// TIA Portal project "Esempio_TCP" (V15.1)

(* hardware
DEVICE "S7-1200 station_2"  S7-1200 Station
   slot 0: "Telaio di montaggio_0"  S7-1200 Rack  Rack  V1.0
   slot 1: "Passivo"  CPU 1214C DC/DC/DC  6ES7 214-1AG40-0XB0  V4.2
DEVICE "S7-1200 station_1"  S7-1200 Station
   slot 0: "Telaio di montaggio_0"  S7-1200 Rack  Rack  V1.0
   slot 1: "Attivo"  CPU 1214C DC/DC/DC  6ES7 214-1AG40-0XB0  V4.2
*)

// ===== PLC "Attivo"  CPU 1214C DC/DC/DC =====

VAR_GLOBAL   // PLC tag table "Tabella delle variabili standard"
   "connetti" AT %I0.0 : Bool;
   "Connesso" AT %M0.0 : Bool;
   "Disconnetti" AT %I0.1 : Bool;
   "invia_dati" AT %I0.2 : Bool;
END_VAR

DATA_BLOCK "Send_block"   // DB4
{ S7_Optimized_Access := 'FALSE' }
VERSION : 0.1
   VAR
      testBool : Bool;
      testInt : Int;
   END_VAR
BEGIN
END_DATA_BLOCK

DATA_BLOCK "Receive_block"   // DB7
{ S7_Optimized_Access := 'FALSE' }
VERSION : 0.1
   VAR
      testBool : Bool;
      testInt : Int;
   END_VAR
BEGIN
END_DATA_BLOCK

// folder: System blocks/Program resources

DATA_BLOCK "Attivo_Connection_DB"   // DB2
{ S7_Optimized_Access := 'TRUE' }
AUTHOR : SIMATIC
FAMILY : MC7Plus
NAME : TC_IP_v4
VERSION : 1.0
// stored: InstanceOfName TCON_IP_v4
"TCON_IP_v4"
BEGIN
   ID := 1;
   InterfaceId := 64;
   RemotePort := 2000;
   ActiveEstablished := true;
   RemoteAddress.ADDR[1] := 192;
   RemoteAddress.ADDR[2] := 168;
   RemoteAddress.ADDR[4] := 2;
END_DATA_BLOCK

// folder: (top level)

ORGANIZATION_BLOCK "Main"   // OB1, LAD, ProgramCycle
TITLE = "Main Program Sweep (Cycle)"
{ S7_Optimized_Access := 'TRUE' }
VERSION : 0.1
   VAR_INPUT
      Initial_Call : Bool;   // Initial call of this OB
      Remanence : Bool;   // =True, if remanent data are available
   END_VAR
   VAR_TEMP
      temp1 : Bool;
      temp2 : Bool;
      temp3 : Bool;
   END_VAR
   VAR_TEMP   // added for the SCL form of the ladder/FBD networks
      _w1 : Bool;
   END_VAR
BEGIN

REGION Network 1
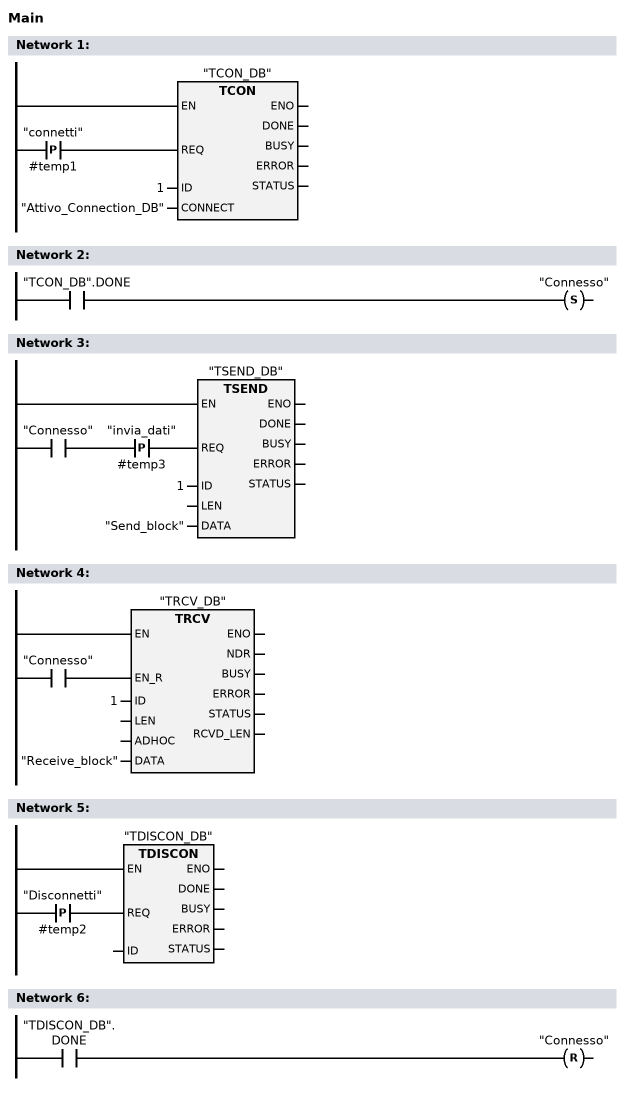
   #_w1 := "connetti" AND NOT #temp1;   // rising edge of "connetti"
   #temp1 := "connetti";
   "TCON_DB"(REQ := #_w1, ID := 1, CONNECT := "Attivo_Connection_DB");   // TCON
END_REGION

REGION Network 2
   RUNG wire#powerrail
      Contact( "TCON_DB".DONE )
      S_Coil( "Connesso" )
   END_RUNG
   // the same network as SCL:
   IF "TCON_DB".DONE THEN "Connesso" := TRUE; END_IF;
END_REGION

REGION Network 3
   #_w1 := "Connesso" AND "invia_dati" AND NOT #temp3;   // rising edge of "invia_dati"
   #temp3 := "invia_dati";
   "TSEND_DB"(REQ := #_w1, ID := 1, DATA := "Send_block");   // TSEND
END_REGION

REGION Network 4
   "TRCV_DB"(EN_R := "Connesso", ID := 1, DATA := "Receive_block");   // TRCV
END_REGION

REGION Network 5
   #_w1 := "Disconnetti" AND NOT #temp2;   // rising edge of "Disconnetti"
   #temp2 := "Disconnetti";
   "TDISCON_DB"(REQ := #_w1);   // TDISCON
END_REGION

REGION Network 6
   RUNG wire#powerrail
      Contact( "TDISCON_DB".DONE )
      R_Coil( "Connesso" )
   END_RUNG
   // the same network as SCL:
   IF "TDISCON_DB".DONE THEN "Connesso" := FALSE; END_IF;
END_REGION
END_ORGANIZATION_BLOCK

// ===== PLC "Passivo"  CPU 1214C DC/DC/DC =====

VAR_GLOBAL   // PLC tag table "Tabella delle variabili standard"
   "Connesso" AT %M0.0 : Bool;
   "Disconnetti" AT %I0.1 : Bool;
   "ApriPorta" AT %I0.0 : Bool;
END_VAR

DATA_BLOCK "Receive_block"   // DB4
{ S7_Optimized_Access := 'FALSE' }
VERSION : 0.1
   VAR
      testBool : Bool;
      testInt : Int;
   END_VAR
BEGIN
END_DATA_BLOCK

// folder: System blocks/Program resources

DATA_BLOCK "Passivo_Connection_DB"   // DB1
{ S7_Optimized_Access := 'TRUE' }
AUTHOR : SIMATIC
FAMILY : MC7Plus
NAME : TC_IP_v4
VERSION : 1.0
// stored: InstanceOfName TCON_IP_v4
"TCON_IP_v4"
BEGIN
   ID := 1;
   InterfaceId := 64;
   LocalPort := 2000;
   RemoteAddress.ADDR[1] := 192;
   RemoteAddress.ADDR[2] := 168;
   RemoteAddress.ADDR[4] := 1;
END_DATA_BLOCK

// folder: (top level)

ORGANIZATION_BLOCK "Main"   // OB1, LAD, ProgramCycle
TITLE = "Main Program Sweep (Cycle)"
{ S7_Optimized_Access := 'TRUE' }
VERSION : 0.1
   VAR_INPUT
      Initial_Call : Bool;   // Initial call of this OB
      Remanence : Bool;   // =True, if remanent data are available
   END_VAR
   VAR_TEMP
      temp1 : Bool;
      temp2 : Bool;
   END_VAR
   VAR_TEMP   // added for the SCL form of the ladder/FBD networks
      _w1 : Bool;
   END_VAR
BEGIN

REGION Network 1
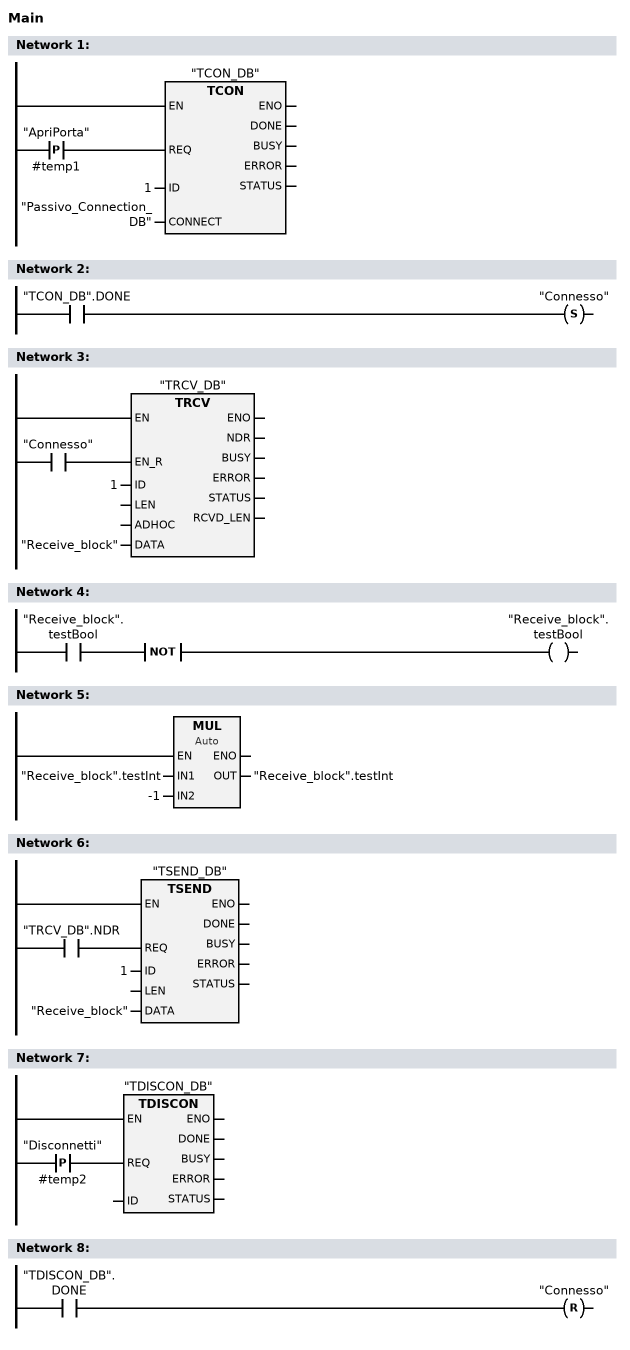
   #_w1 := "ApriPorta" AND NOT #temp1;   // rising edge of "ApriPorta"
   #temp1 := "ApriPorta";
   "TCON_DB"(REQ := #_w1, ID := 1, CONNECT := "Passivo_Connection_DB");   // TCON
END_REGION

REGION Network 2
   RUNG wire#powerrail
      Contact( "TCON_DB".DONE )
      S_Coil( "Connesso" )
   END_RUNG
   // the same network as SCL:
   IF "TCON_DB".DONE THEN "Connesso" := TRUE; END_IF;
END_REGION

REGION Network 3
   "TRCV_DB"(EN_R := "Connesso", ID := 1, DATA := "Receive_block");   // TRCV
END_REGION

REGION Network 4
   RUNG wire#powerrail
      Contact( "Receive_block".testBool )
      Not()
      Coil( "Receive_block".testBool )
   END_RUNG
   // the same network as SCL:
   "Receive_block".testBool := NOT "Receive_block".testBool;
END_REGION

REGION Network 5
   RUNG wire#powerrail
      Mul(in1 := "Receive_block".testInt, in2 := -1, out => "Receive_block".testInt)
   END_RUNG
   // the same network as SCL:
   "Receive_block".testInt := "Receive_block".testInt * (-1);
END_REGION

REGION Network 6
   "TSEND_DB"(REQ := "TRCV_DB".NDR, ID := 1, DATA := "Receive_block");   // TSEND
END_REGION

REGION Network 7
   #_w1 := "Disconnetti" AND NOT #temp2;   // rising edge of "Disconnetti"
   #temp2 := "Disconnetti";
   "TDISCON_DB"(REQ := #_w1);   // TDISCON
END_REGION

REGION Network 8
   RUNG wire#powerrail
      Contact( "TDISCON_DB".DONE )
      R_Coil( "Connesso" )
   END_RUNG
   // the same network as SCL:
   IF "TDISCON_DB".DONE THEN "Connesso" := FALSE; END_IF;
END_REGION
END_ORGANIZATION_BLOCK